FUNCTION_BLOCK TRAY_HMI (* Basic Function Block Type *)
  (* Standard: 61499-2 *)
  (* Version 0.2, 2003-12-04, JHC, Rockwell Automation, Renamed for better indexing. *)
  (* Version 0.1, 2002-11-05, JHC, Rockwell Automation, Corrected missing ST element in Algorithm REQ. *)
  (* Version 0.0, 2000-05-30, JHC, Rockwell Automation *)
  (* Compiler header: package fb.rt.pnp; *)
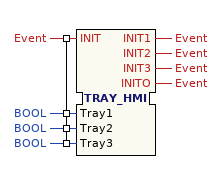
  EVENT_INPUT
    INIT WITH Tray1, Tray2, Tray3; (* Initialization Request *)
  END_EVENT
  EVENT_OUTPUT
    INIT1; (* Initialization Confirm *)
    INIT2;
    INIT3;
    INITO;
  END_EVENT
  VAR_INPUT
    Tray1 : BOOL; (* Input event qualifier *)
    Tray2 : BOOL;
    Tray3 : BOOL;
  END_VAR
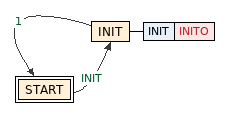
  EC_STATES
    START; (* Initial State *)
    INIT : INIT -> INITO; (* Initialization *)
  END_STATES
  EC_TRANSITIONS
    START TO INIT := INIT;
    INIT TO START := 1;
  END_TRANSITIONS
  ALGORITHM INIT IN Java:
if (Tray1.value)
{
   INIT1.serviceEvent(this);
}
if (Tray2.value)
{
   INIT2.serviceEvent(this);
}
if (Tray3.value)
{
   INIT3.serviceEvent(this);
}
  END_ALGORITHM
END_FUNCTION_BLOCK
